# EPICS autosave request: iocBoot/sioc-li24-im01/adc_manual.req
file "manual.req" AREA=LI24,POS=708
file "manual.req" AREA=LI25,POS=236
